TYPE ST_OneProcessServoPara :
    STRUCT
        Position :LREAL;
        Velocity :LREAL;
        Distance :LREAL;
        ACC      :LREAL;
        DEC      :LREAL;
        Jerk     :LREAL;
    END_STRUCT
END_TYPE

(* stored: Version 1.1.0.1, ProductVersion 3.1.4024.13
   DUT ST_OneProcessServoPara: Id {ec7b37b7-2cee-4531-b3bc-97c8c08a025d} *)
